TYPE ST_WcState :
STRUCT
	WcState		: BIT;
	InputToggle	: BIT;
END_STRUCT
END_TYPE

(* stored: Version 1.1.0.1, ProductVersion 3.1.4024.3
   DUT ST_WcState: Id {d7c168e5-30b2-0bc0-37ca-0860f9943a1c} *)
